{attribute addProperty BoxType "EJ7334-0008-0016"}
{attribute addProperty Id "StatusAT %I*Status_7570E3BD162"}
{attribute addProperty CRC "3688950303"}
{attribute addProperty SizeInBites "16"}
{attribute addProperty SizeInBytes "2"}
TYPE DCM_Status_Channel_DBE0EA1F :
STRUCT
	{attribute addProperty Name "Status"}
	Status AT %I* : Status_7570E3BD;
END_STRUCT
END_TYPE

(* stored: Version 1.2.0.0, ProductVersion 3.1.4024.9
   DUT DCM_Status_Channel_DBE0EA1F: Id {5c8320f9-9e74-4e89-ba0f-0a2c3039e11f} *)
